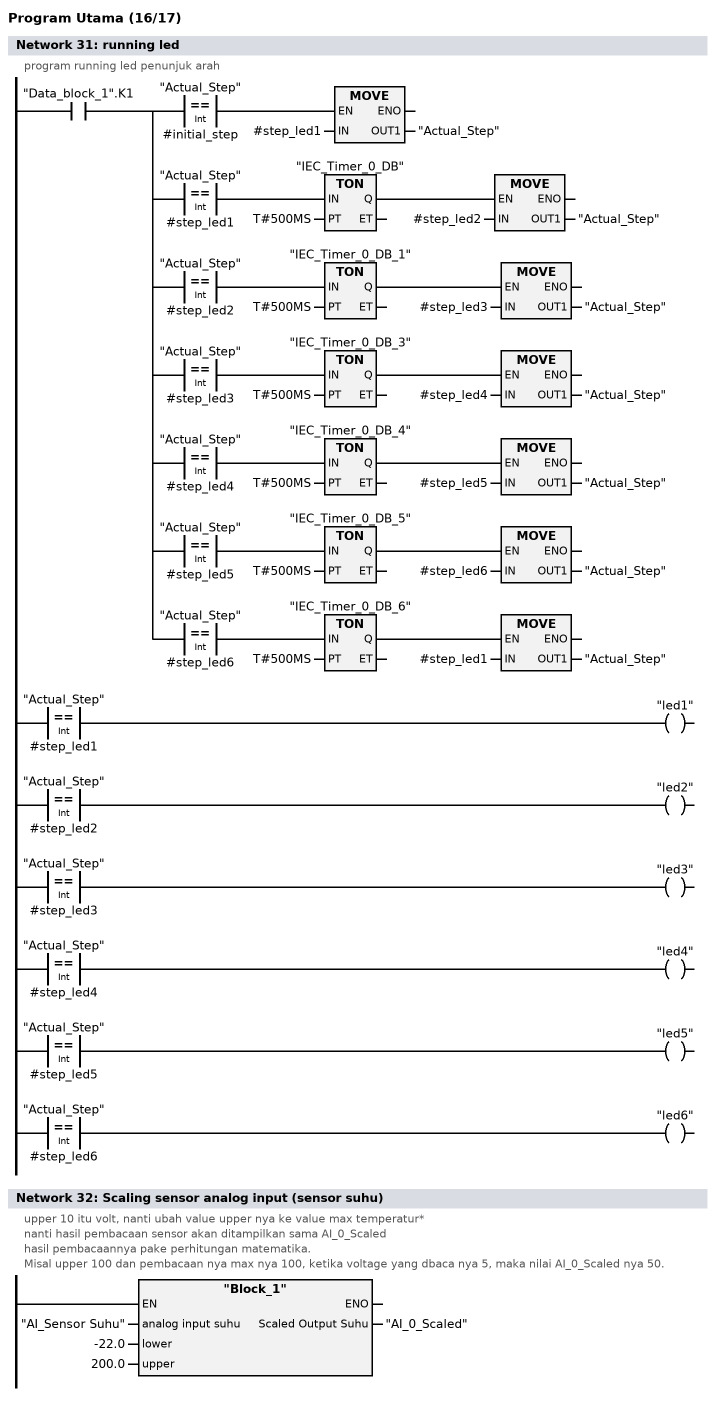
   IF "Data_block_1".K1 AND ("Actual_Step" = #initial_step) THEN "Actual_Step" := #step_led1; END_IF;
   "IEC_Timer_0_DB".TON(IN := "Data_block_1".K1 AND ("Actual_Step" = #step_led1), PT := T#500MS);
   IF "IEC_Timer_0_DB".Q THEN "Actual_Step" := #step_led2; END_IF;
   "IEC_Timer_0_DB_1".TON(IN := "Data_block_1".K1 AND ("Actual_Step" = #step_led2), PT := T#500MS);
   IF "IEC_Timer_0_DB_1".Q THEN "Actual_Step" := #step_led3; END_IF;
   "IEC_Timer_0_DB_3".TON(IN := "Data_block_1".K1 AND ("Actual_Step" = #step_led3), PT := T#500MS);
   IF "IEC_Timer_0_DB_3".Q THEN "Actual_Step" := #step_led4; END_IF;
   "IEC_Timer_0_DB_4".TON(IN := "Data_block_1".K1 AND ("Actual_Step" = #step_led4), PT := T#500MS);
   IF "IEC_Timer_0_DB_4".Q THEN "Actual_Step" := #step_led5; END_IF;
   "IEC_Timer_0_DB_5".TON(IN := "Data_block_1".K1 AND ("Actual_Step" = #step_led5), PT := T#500MS);
   IF "IEC_Timer_0_DB_5".Q THEN "Actual_Step" := #step_led6; END_IF;
   "IEC_Timer_0_DB_6".TON(IN := "Data_block_1".K1 AND ("Actual_Step" = #step_led6), PT := T#500MS);
   IF "IEC_Timer_0_DB_6".Q THEN "Actual_Step" := #step_led1; END_IF;
   "led1" := "Actual_Step" = #step_led1;
   "led2" := "Actual_Step" = #step_led2;
   "led3" := "Actual_Step" = #step_led3;
   "led4" := "Actual_Step" = #step_led4;
   "led5" := "Actual_Step" = #step_led5;
   "led6" := "Actual_Step" = #step_led6;
END_REGION

REGION Network 32: Scaling sensor analog input (sensor suhu)
   // upper 10 itu volt, nanti ubah value upper nya ke value max temperatur* 
   // nanti hasil pembacaan sensor akan ditampilkan sama AI_0_Scaled
   // hasil pembacaannya pake perhitungan matematika. 
   // Misal upper 100 dan pembacaan nya max nya 100, ketika voltage yang dbaca nya 5, maka nilai AI_0_Scaled nya 50.
   RUNG wire#powerrail
      "Block_1"("analog input suhu" := "AI_Sensor Suhu", lower := -22.0, upper := 200.0, "Scaled Output Suhu" => "AI_0_Scaled")
   END_RUNG
   // the same network as SCL:
   "Block_1"("analog input suhu" := "AI_Sensor Suhu",
             lower := -22.0,
             upper := 200.0,
             "Scaled Output Suhu" => "AI_0_Scaled");
END_REGION

REGION Network 33: Data memory suhu kanan
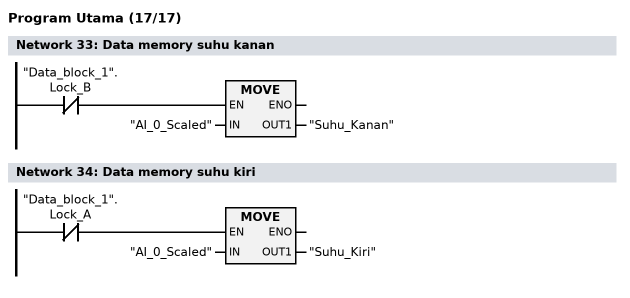
   RUNG wire#powerrail
      I_Contact( "Data_block_1".Lock_B )
      Move(in := "AI_0_Scaled", out1 => "Suhu_Kanan")
   END_RUNG
   // the same network as SCL:
   IF NOT "Data_block_1".Lock_B THEN "Suhu_Kanan" := "AI_0_Scaled"; END_IF;
END_REGION

REGION Network 34: Data memory suhu kiri
   RUNG wire#powerrail
      I_Contact( "Data_block_1".Lock_A )
      Move(in := "AI_0_Scaled", out1 => "Suhu_Kiri")
   END_RUNG
   // the same network as SCL:
   IF NOT "Data_block_1".Lock_A THEN "Suhu_Kiri" := "AI_0_Scaled"; END_IF;
END_REGION
END_ORGANIZATION_BLOCK

(* ===== HMI "HMI_RT_1" =====
system functions are stored by id; their names below are inferred from use
connection "Connection_1": ETHERNET, S7_1200_OMS
connection "HMI_Connection_1": ETHERNET, S7_1200_OMS

HMI tags "Default tag table"
   "prox_a" : Bool = PLC prox_a1 AT %I0.0, 1 s
   "prox_b" : Bool = PLC prox_b1 AT %I0.1, 1 s
   "Q1" : Bool = PLC "Q1-1" AT %M0.0, 1 s
   "Q2" : Bool = PLC "Q2-1" AT %M0.1, 1 s
   "du_a" : Bool = PLC du_a AT %M0.2, 1 s
   "dd_b" : Bool = PLC dd_b AT %M0.3, 1 s
   "k_proxa" : Bool = PLC k_proxa AT %M0.4, 1 s
   "k_proxb" : Bool = PLC k_proxb AT %M0.5, 1 s
   "counter" : Bool = PLC counter AT %M0.6, 1 s
   "pemutus" : Bool = PLC pemutus AT %M0.7, 1 s
   "du_b" : Bool = PLC "ProxA+" AT %M1.0, 1 s
   "dd_a" : Bool = PLC "ProxB-" AT %M1.1, 1 s
   "reset" : Bool = PLC reset AT %M1.2, 1 s
   "Clock_Byte" : Byte = PLC Clock_Byte AT %MB10, 1 s
   "Clock_10Hz" : Bool = PLC Clock_10Hz AT %M10.0, 1 s
   "Clock_5Hz" : Bool = PLC Clock_5Hz AT %M10.1, 1 s
   "Clock_2.5Hz" : Bool = PLC "Clock_2.5Hz" AT %M10.2, 1 s
   "Clock_2Hz" : Bool = PLC Clock_2Hz AT %M10.3, 1 s
   "Clock_1.25Hz" : Bool = PLC "Clock_1.25Hz" AT %M10.4, 1 s
   "Clock_1Hz" : Bool = PLC Clock_1Hz AT %M10.5, 1 s
   "Clock_0.625Hz" : Bool = PLC "Clock_0.625Hz" AT %M10.6, 1 s
   "Clock_0.5Hz" : Bool = PLC "Clock_0.5Hz" AT %M10.7, 1 s
   "System_Byte" : Byte = PLC System_Byte AT %MB100, 1 s
   "FirstScan" : Bool = PLC FirstScan AT %M100.0, 1 s
   "DiagStatusUpdate" : Bool = PLC DiagStatusUpdate AT %M100.1, 1 s
   "AlwaysTRUE" : Bool = PLC AlwaysTRUE AT %M100.2, 1 s
   "AlwaysFALSE" : Bool = PLC AlwaysFALSE AT %M100.3, 1 s
   "Data_block_1_dataroda1{0}" : Real = PLC Data_block_1.dataroda1[0] AT %DB3.DBD21370, 1 s
   "Data_block_1_dataroda1{1}" : Real = PLC Data_block_1.dataroda1[1] AT %DB3.DBD21374, 1 s
   "Data_block_1_dataroda1{2}" : Real = PLC Data_block_1.dataroda1[2] AT %DB3.DBD21378, 1 s
   "Data_block_1_dataroda1{3}" : Real = PLC Data_block_1.dataroda1[3] AT %DB3.DBD21382, 1 s

screen "Screen_1" 1024x768
   on GenerateScreen: function_bb0abc73()
   Switch "Switch_1" at 110,0 size 120x88; CaptionText 'a'; TextOff 'OFF'; TextOn 'ON'
      ProcessValue <- "prox_a"
   Switch "Switch_2" at 256,0 size 120x88; CaptionText 'b'; TextOff 'OFF'; TextOn 'ON'
      ProcessValue <- "prox_b"
   StatusForce "Watch table_1" at 49,111 size 600x300; ToolTipText 'Text'
*)